DATA_BLOCK "DB2001_EA"
TITLE = DB2001_EA
{ S7_Optimized_Access := 'FALSE' }
AUTHOR : ABH
FAMILY : ZeusControl
VERSION : 1.0
//Bloque de datos entrada analogica
   STRUCT
      EA { S7_SetPoint := 'False'} : Array[0.."N_MAX_DISP_EA"] of "UDT_ZC_DISP_EA";
      Mux { S7_SetPoint := 'False'} : Array[0.."N_MAX_MUX_DISP"] of "UDT_ZC_DISP_MUX_EA";
      Agrup : Array[0.."N_MAX_DISP_AGRUP"] of "UDT_ZC_DISP_AGRUP";
   END_STRUCT;


BEGIN
   EA[0].Hmi_Estado := 0;
   EA[0].Estado_ValorIngenieria := 0.0;
   EA[0].Estado_AutoMan := FALSE;
   EA[0].Alarmas_Min := FALSE;
   EA[0].Alarmas_Max := FALSE;
   EA[0].Alarmas_HiloRoto := FALSE;
   EA[0].Alarmas_Lectura := FALSE;
   EA[0].Alarmas_Parametros := FALSE;
   EA[0].Alarmas_General := FALSE;
   EA[0].Config_Habilitar := FALSE;
   EA[0].Config_HabilitarAlarmaMin := FALSE;
   EA[0].Config_HabilitarAlarmaMax := FALSE;
   EA[0].Config_HisteresisTipo := FALSE;
   EA[0].Config_HabilitarEscalado := TRUE;
   EA[0].Aux_oldAlarma := FALSE;
   EA[0].Aux_oldAutoMan := FALSE;
   EA[0].Config_GrupoAlarma := 0;
   EA[0].Estado_ValorTarjeta := 0;
   EA[0].Estado_Lectura := 16#0000;
   EA[0].Orden_ConsignaManual := 0.0;
   EA[0].Config_DireccionEntradaByte := 0;
   EA[0].Config_EscaladoMinTarjeta := 0;
   EA[0].Config_EscaladoMaxTarjeta := 27648;
   EA[0].Config_EscaladoMinIngenieria := 0.0;
   EA[0].Config_EscaladoMaxIngenieria := 100.0;
   EA[0].Config_EscaladoOffset := 0.0;
   EA[0].Config_ErrorMinIngenieria := 0.0;
   EA[0].Config_ErrorMaxIngenieria := 100.0;
   EA[0].Config_ErrorMinHisteresis := 0.0;
   EA[0].Config_ErrorMaxHisteresis := 0.0;
   EA[0].Aux_Estado := 0;
   EA[1].Hmi_Estado := 1;
   EA[1].Estado_ValorIngenieria := 28.02083;
   EA[1].Estado_AutoMan := FALSE;
   EA[1].Alarmas_Min := FALSE;
   EA[1].Alarmas_Max := FALSE;
   EA[1].Alarmas_HiloRoto := FALSE;
   EA[1].Alarmas_Lectura := FALSE;
   EA[1].Alarmas_Parametros := FALSE;
   EA[1].Alarmas_General := FALSE;
   EA[1].Config_Habilitar := TRUE;
   EA[1].Config_HabilitarAlarmaMin := FALSE;
   EA[1].Config_HabilitarAlarmaMax := FALSE;
   EA[1].Config_HisteresisTipo := FALSE;
   EA[1].Config_HabilitarEscalado := TRUE;
   EA[1].Aux_oldAlarma := FALSE;
   EA[1].Aux_oldAutoMan := FALSE;
   EA[1].Config_GrupoAlarma := 0;
   EA[1].Estado_ValorTarjeta := 6570;
   EA[1].Estado_Lectura := 16#0000;
   EA[1].Orden_ConsignaManual := 28.02083;
   EA[1].Config_DireccionEntradaByte := 2100;
   EA[1].Config_EscaladoMinTarjeta := 0;
   EA[1].Config_EscaladoMaxTarjeta := 27648;
   EA[1].Config_EscaladoMinIngenieria := -10.0;
   EA[1].Config_EscaladoMaxIngenieria := 150.0;
   EA[1].Config_EscaladoOffset := 0.0;
   EA[1].Config_ErrorMinIngenieria := 0.0;
   EA[1].Config_ErrorMaxIngenieria := 100.0;
   EA[1].Config_ErrorMinHisteresis := 0.0;
   EA[1].Config_ErrorMaxHisteresis := 0.0;
   EA[1].Aux_Estado := 1;
   Mux[0].Habilitar := TRUE;
   Mux[0].ExisteCambio := FALSE;
   Mux[0].MaxVisible := FALSE;
   Mux[0].Index := 10;
   Mux[0].oldIndex := 10;
   Mux[0].EA.Hmi_Estado := 1;
   Mux[0].EA.Estado_ValorIngenieria := -30.0;
   Mux[0].EA.Estado_AutoMan := FALSE;
   Mux[0].EA.Alarmas_Min := FALSE;
   Mux[0].EA.Alarmas_Max := FALSE;
   Mux[0].EA.Alarmas_HiloRoto := FALSE;
   Mux[0].EA.Alarmas_Lectura := FALSE;
   Mux[0].EA.Alarmas_Parametros := FALSE;
   Mux[0].EA.Alarmas_General := FALSE;
   Mux[0].EA.Config_Habilitar := TRUE;
   Mux[0].EA.Config_HabilitarAlarmaMin := FALSE;
   Mux[0].EA.Config_HabilitarAlarmaMax := FALSE;
   Mux[0].EA.Config_HisteresisTipo := FALSE;
   Mux[0].EA.Config_HabilitarEscalado := FALSE;
   Mux[0].EA.Aux_oldAlarma := FALSE;
   Mux[0].EA.Aux_oldAutoMan := FALSE;
   Mux[0].EA.Config_GrupoAlarma := 0;
   Mux[0].EA.Estado_ValorTarjeta := 0;
   Mux[0].EA.Estado_Lectura := 16#0000;
   Mux[0].EA.Orden_ConsignaManual := 30.0;
   Mux[0].EA.Config_DireccionEntradaByte := 3120;
   Mux[0].EA.Config_EscaladoMinTarjeta := 0;
   Mux[0].EA.Config_EscaladoMaxTarjeta := 27648;
   Mux[0].EA.Config_EscaladoMinIngenieria := 0.0;
   Mux[0].EA.Config_EscaladoMaxIngenieria := 50000.0;
   Mux[0].EA.Config_EscaladoOffset := 2.0;
   Mux[0].EA.Config_ErrorMinIngenieria := 0.0;
   Mux[0].EA.Config_ErrorMaxIngenieria := 100.0;
   Mux[0].EA.Config_ErrorMinHisteresis := 0.0;
   Mux[0].EA.Config_ErrorMaxHisteresis := 0.0;
   Mux[0].EA.Aux_Estado := 1;
   Mux[1].Habilitar := TRUE;
   Mux[1].ExisteCambio := FALSE;
   Mux[1].MaxVisible := FALSE;
   Mux[1].Index := 0;
   Mux[1].oldIndex := 0;
   Mux[1].EA.Hmi_Estado := 0;
   Mux[1].EA.Estado_ValorIngenieria := 0.0;
   Mux[1].EA.Estado_AutoMan := FALSE;
   Mux[1].EA.Alarmas_Min := FALSE;
   Mux[1].EA.Alarmas_Max := FALSE;
   Mux[1].EA.Alarmas_HiloRoto := FALSE;
   Mux[1].EA.Alarmas_Lectura := FALSE;
   Mux[1].EA.Alarmas_Parametros := FALSE;
   Mux[1].EA.Alarmas_General := FALSE;
   Mux[1].EA.Config_Habilitar := FALSE;
   Mux[1].EA.Config_HabilitarAlarmaMin := FALSE;
   Mux[1].EA.Config_HabilitarAlarmaMax := FALSE;
   Mux[1].EA.Config_HisteresisTipo := FALSE;
   Mux[1].EA.Config_HabilitarEscalado := TRUE;
   Mux[1].EA.Aux_oldAlarma := FALSE;
   Mux[1].EA.Aux_oldAutoMan := FALSE;
   Mux[1].EA.Config_GrupoAlarma := 0;
   Mux[1].EA.Estado_ValorTarjeta := 0;
   Mux[1].EA.Estado_Lectura := 16#0000;
   Mux[1].EA.Orden_ConsignaManual := 0.0;
   Mux[1].EA.Config_DireccionEntradaByte := 0;
   Mux[1].EA.Config_EscaladoMinTarjeta := 0;
   Mux[1].EA.Config_EscaladoMaxTarjeta := 27648;
   Mux[1].EA.Config_EscaladoMinIngenieria := 0.0;
   Mux[1].EA.Config_EscaladoMaxIngenieria := 100.0;
   Mux[1].EA.Config_EscaladoOffset := 0.0;
   Mux[1].EA.Config_ErrorMinIngenieria := 0.0;
   Mux[1].EA.Config_ErrorMaxIngenieria := 100.0;
   Mux[1].EA.Config_ErrorMinHisteresis := 0.0;
   Mux[1].EA.Config_ErrorMaxHisteresis := 0.0;
   Mux[1].EA.Aux_Estado := 0;
   Agrup[0].AlgunaEnManual := FALSE;
   Agrup[0].AlgunaAlarma := FALSE;
   Agrup[0].NuevaAlarma := FALSE;
   Agrup[1].AlgunaEnManual := FALSE;
   Agrup[1].AlgunaAlarma := FALSE;
   Agrup[1].NuevaAlarma := FALSE;

END_DATA_BLOCK

